TYPE ST_ZoneAlarmStatus :
STRUCT
    bOkToRun : BOOL;           
    nHighestSeverity : UINT;   
END_STRUCT
END_TYPE

(* stored: Version 1.1.0.1, ProductVersion 3.1.4026.11
   DUT ST_ZoneAlarmStatus: Id {667a1402-e997-4e2e-8691-3d80689897d4} *)
